SUBAPPLICATION Uebung_072_AUI (* GBSD und WBSD auf UT ausgeben (Adapter Version) *)
  (* Standard: 61499-2; Description: Copyright (c) 2023 Meisterschulen am Ostbahnhof This program and the accompanying materials are made available under the terms of the Eclipse Public License 2.0 which is available at https://www.eclipse.org/legal/epl-2.0/ SPDX-License-Identifier: EPL-2.0 *)
  (* Version 1.0, 2026-04-19, Franz Höpfinger, Meisterschulen am Ostbahnhof, initial API and implementation (Adapter Version of Uebung_072) *)
  PACKAGE Uebungen;
  IMPORT Uebungen::const::UT::TECU::DefaultPool_TECU::NumberVariable_Ground_based_machine_speed;
  IMPORT Uebungen::const::UT::TECU::DefaultPool_TECU::NumberVariable_Wheel_based_machine_speed;
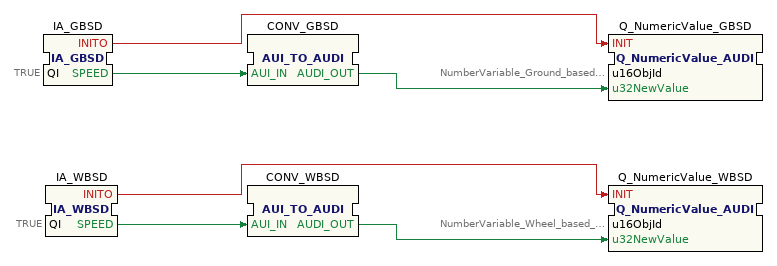
  FBS
    IA_GBSD : isobus::tecu::IA_GBSD(QI := TRUE);
    Q_NumericValue_GBSD : isobus::UT::Q::Q_NumericValue_AUDI(u16ObjId := NumberVariable_Ground_based_machine_speed);
    IA_WBSD : isobus::tecu::IA_WBSD(QI := TRUE);
    Q_NumericValue_WBSD : isobus::UT::Q::Q_NumericValue_AUDI(u16ObjId := NumberVariable_Wheel_based_machine_speed);
    CONV_GBSD : adapter::conversion::unidirectional::AUI_TO_AUDI;
    CONV_WBSD : adapter::conversion::unidirectional::AUI_TO_AUDI;
  END_FBS
  EVENT_CONNECTIONS
    IA_GBSD.INITO TO Q_NumericValue_GBSD.INIT;
    IA_WBSD.INITO TO Q_NumericValue_WBSD.INIT;
  END_CONNECTIONS
  ADAPTER_CONNECTIONS
    IA_GBSD.SPEED TO CONV_GBSD.AUI_IN;
    CONV_GBSD.AUDI_OUT TO Q_NumericValue_GBSD.u32NewValue;
    IA_WBSD.SPEED TO CONV_WBSD.AUI_IN;
    CONV_WBSD.AUDI_OUT TO Q_NumericValue_WBSD.u32NewValue;
  END_CONNECTIONS
END_SUBAPPLICATION
